ABB RAPID module: Module1.mod

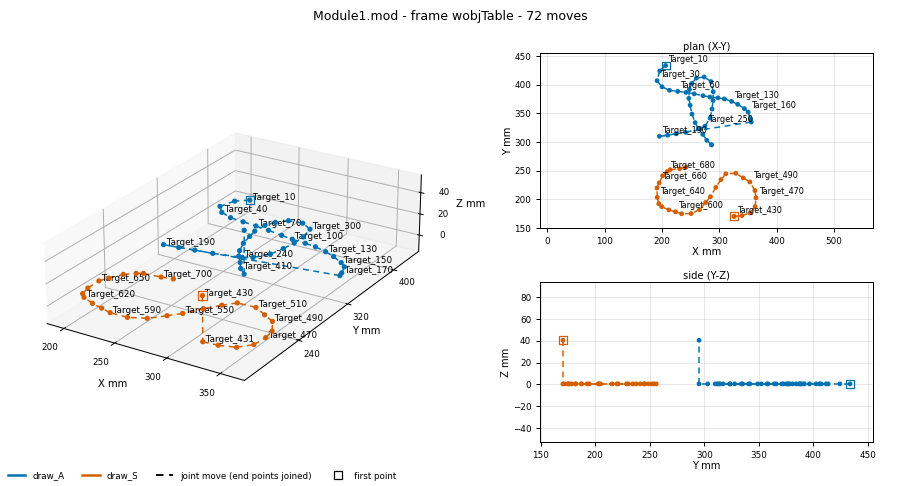
[picture p0: tool path of Module1.mod in frame wobjTable, 72 of 76 moves have a stored position in this frame; points joined in program order, loops and branches not executed]
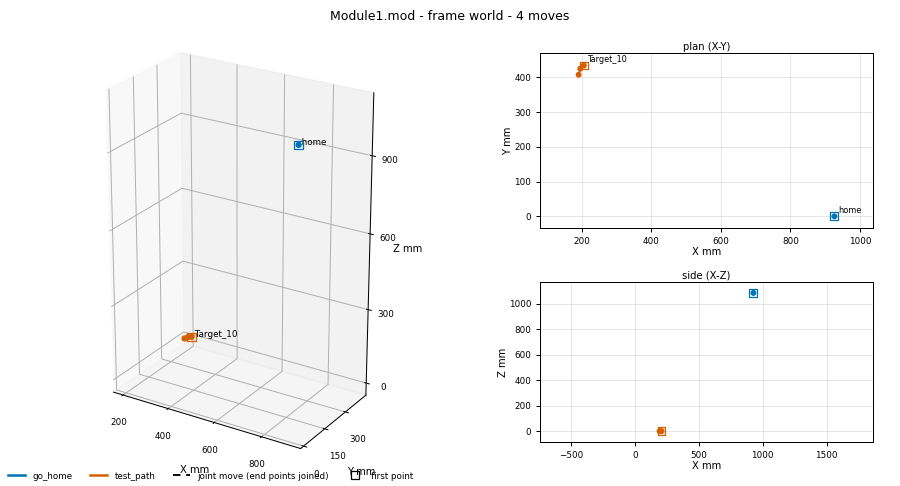
[picture p1: tool path of Module1.mod in frame world, 4 of 76 moves have a stored position in this frame; points joined in program order, loops and branches not executed]
MODULE Module1
	CONST robtarget home:=[[926.669182372,0,1084.5],[0.5,0,0.866025404,0],[0,0,0,0],[9E+09,9E+09,9E+09,9E+09,9E+09,9E+09]];
	CONST robtarget Target_10:=[[206.293,433.63,0.5],[0,0,1,0],[0,0,0,0],[9E+09,9E+09,9E+09,9E+09,9E+09,9E+09]];
	CONST robtarget Target_20:=[[196.05,424.338,0.5],[0,0,1,0],[0,0,0,0],[9E+09,9E+09,9E+09,9E+09,9E+09,9E+09]];
	CONST robtarget Target_30:=[[191.33,407.149,0.5],[0,0,1,0],[0,0,0,0],[9E+09,9E+09,9E+09,9E+09,9E+09,9E+09]];
	CONST robtarget Target_40:=[[200.077,396.45,0.5],[0,0,1,0],[0,0,0,0],[9E+09,9E+09,9E+09,9E+09,9E+09,9E+09]];
	CONST robtarget Target_50:=[[213.027,390.387,0.5],[0,0,1,0],[0,0,0,0],[9E+09,9E+09,9E+09,9E+09,9E+09,9E+09]];
	CONST robtarget Target_60:=[[227.402,388.502,0.5],[0,0,1,0],[0,0,0,0],[9E+09,9E+09,9E+09,9E+09,9E+09,9E+09]];
	CONST robtarget Target_70:=[[241.792,386.616,0.5],[0,0,1,0],[0,0,0,0],[9E+09,9E+09,9E+09,9E+09,9E+09,9E+09]];
	CONST robtarget Target_80:=[[256.194,384.262,0.5],[0,0,1,0],[0,0,0,0],[9E+09,9E+09,9E+09,9E+09,9E+09,9E+09]];
	CONST robtarget Target_90:=[[271.536,380.972,0.5],[0,0,1,0],[0,0,0,0],[9E+09,9E+09,9E+09,9E+09,9E+09,9E+09]];
	CONST robtarget Target_100:=[[283.637,378.618,0.5],[0,0,1,0],[0,0,0,0],[9E+09,9E+09,9E+09,9E+09,9E+09,9E+09]];
	CONST robtarget Target_110:=[[297.618,377.191,0.5],[0,0,1,0],[0,0,0,0],[9E+09,9E+09,9E+09,9E+09,9E+09,9E+09]];
	CONST robtarget Target_120:=[[308.809,375.301,0.5],[0,0,1,0],[0,0,0,0],[9E+09,9E+09,9E+09,9E+09,9E+09,9E+09]];
	CONST robtarget Target_130:=[[321.398,371.074,0.5],[0,0,1,0],[0,0,0,0],[9E+09,9E+09,9E+09,9E+09,9E+09,9E+09]];
	CONST robtarget Target_140:=[[332.122,365.914,0.5],[0,0,1,0],[0,0,0,0],[9E+09,9E+09,9E+09,9E+09,9E+09,9E+09]];
	CONST robtarget Target_150:=[[343.779,358.412,0.5],[0,0,1,0],[0,0,0,0],[9E+09,9E+09,9E+09,9E+09,9E+09,9E+09]];
	CONST robtarget Target_160:=[[350.301,352.321,0.5],[0,0,1,0],[0,0,0,0],[9E+09,9E+09,9E+09,9E+09,9E+09,9E+09]];
	CONST robtarget Target_170:=[[354.455,340.628,0.5],[0,0,1,0],[0,0,0,0],[9E+09,9E+09,9E+09,9E+09,9E+09,9E+09]];
	CONST robtarget Target_180:=[[355.831,335.016,0.5],[0,0,1,0],[0,0,0,0],[9E+09,9E+09,9E+09,9E+09,9E+09,9E+09]];
	CONST robtarget Target_190:=[[195.464,310.023,0.5],[0,0,1,0],[0,0,0,0],[9E+09,9E+09,9E+09,9E+09,9E+09,9E+09]];
	CONST robtarget Target_200:=[[209.832,311.96,0.5],[0,0,1,0],[0,0,0,0],[9E+09,9E+09,9E+09,9E+09,9E+09,9E+09]];
	CONST robtarget Target_210:=[[224.671,314.499,0.5],[0,0,1,0],[0,0,0,0],[9E+09,9E+09,9E+09,9E+09,9E+09,9E+09]];
	CONST robtarget Target_220:=[[241.385,317.028,0.5],[0,0,1,0],[0,0,0,0],[9E+09,9E+09,9E+09,9E+09,9E+09,9E+09]];
	CONST robtarget Target_240:=[[267.009,323.298,0.5],[0,0,1,0],[0,0,0,0],[9E+09,9E+09,9E+09,9E+09,9E+09,9E+09]];
	CONST robtarget Target_250:=[[274.99,327.846,0.5],[0,0,1,0],[0,0,0,0],[9E+09,9E+09,9E+09,9E+09,9E+09,9E+09]];
	CONST robtarget Target_260:=[[283.914,341.795,0.5],[0,0,1,0],[0,0,0,0],[9E+09,9E+09,9E+09,9E+09,9E+09,9E+09]];
	CONST robtarget Target_270:=[[287.258,357.634,0.5],[0,0,1,0],[0,0,0,0],[9E+09,9E+09,9E+09,9E+09,9E+09,9E+09]];
	CONST robtarget Target_280:=[[289.199,372.546,0.5],[0,0,1,0],[0,0,0,0],[9E+09,9E+09,9E+09,9E+09,9E+09,9E+09]];
	CONST robtarget Target_290:=[[289.278,387.93,0.5],[0,0,1,0],[0,0,0,0],[9E+09,9E+09,9E+09,9E+09,9E+09,9E+09]];
	CONST robtarget Target_300:=[[285.64,405.649,0.5],[0,0,1,0],[0,0,0,0],[9E+09,9E+09,9E+09,9E+09,9E+09,9E+09]];
	CONST robtarget Target_310:=[[273.566,413.584,0.5],[0,0,1,0],[0,0,0,0],[9E+09,9E+09,9E+09,9E+09,9E+09,9E+09]];
	CONST robtarget Target_320:=[[260.057,411.732,0.5],[0,0,1,0],[0,0,0,0],[9E+09,9E+09,9E+09,9E+09,9E+09,9E+09]];
	CONST robtarget Target_330:=[[252.101,402.428,0.5],[0,0,1,0],[0,0,0,0],[9E+09,9E+09,9E+09,9E+09,9E+09,9E+09]];
	CONST robtarget Target_340:=[[247.861,391.726,0.5],[0,0,1,0],[0,0,0,0],[9E+09,9E+09,9E+09,9E+09,9E+09,9E+09]];
	CONST robtarget Target_350:=[[246.853,376.366,0.5],[0,0,1,0],[0,0,0,0],[9E+09,9E+09,9E+09,9E+09,9E+09,9E+09]];
	CONST robtarget Target_360:=[[249.115,364.257,0.5],[0,0,1,0],[0,0,0,0],[9E+09,9E+09,9E+09,9E+09,9E+09,9E+09]];
	CONST robtarget Target_370:=[[252.292,348.884,0.5],[0,0,1,0],[0,0,0,0],[9E+09,9E+09,9E+09,9E+09,9E+09,9E+09]];
	CONST robtarget Target_380:=[[257.797,333.965,0.5],[0,0,1,0],[0,0,0,0],[9E+09,9E+09,9E+09,9E+09,9E+09,9E+09]];
	CONST robtarget Target_390:=[[263.328,323.698,0.5],[0,0,1,0],[0,0,0,0],[9E+09,9E+09,9E+09,9E+09,9E+09,9E+09]];
	CONST robtarget Target_400:=[[271.19,313.417,0.5],[0,0,1,0],[0,0,0,0],[9E+09,9E+09,9E+09,9E+09,9E+09,9E+09]];
	CONST robtarget Target_410:=[[278.124,303.135,0.5],[0,0,1,0],[0,0,0,0],[9E+09,9E+09,9E+09,9E+09,9E+09,9E+09]];
	CONST robtarget Target_420:=[[286.472,295.172,0.5],[0,0,1,0],[0,0,0,0],[9E+09,9E+09,9E+09,9E+09,9E+09,9E+09]];
	CONST robtarget Target_421:=[[286.472,295.172,40.5],[0,0,1,0],[0,0,0,0],[9E+09,9E+09,9E+09,9E+09,9E+09,9E+09]];
	CONST robtarget Target_430:=[[325.977,170.345,40.5],[0,0,1,0],[0,0,0,0],[9E+09,9E+09,9E+09,9E+09,9E+09,9E+09]];
	CONST robtarget Target_431:=[[325.977,170.345,0.5],[0,0,1,0],[0,0,0,0],[9E+09,9E+09,9E+09,9E+09,9E+09,9E+09]];
	CONST robtarget Target_440:=[[339.546,171.622,0.5],[0,0,1,0],[0,0,0,0],[9E+09,9E+09,9E+09,9E+09,9E+09,9E+09]];
	CONST robtarget Target_450:=[[353.612,176.166,0.5],[0,0,1,0],[0,0,0,0],[9E+09,9E+09,9E+09,9E+09,9E+09,9E+09]];
	CONST robtarget Target_460:=[[362.57,187.303,0.5],[0,0,1,0],[0,0,0,0],[9E+09,9E+09,9E+09,9E+09,9E+09,9E+09]];
	CONST robtarget Target_470:=[[364.055,202.715,0.5],[0,0,1,0],[0,0,0,0],[9E+09,9E+09,9E+09,9E+09,9E+09,9E+09]];
	CONST robtarget Target_480:=[[362.245,215.349,0.5],[0,0,1,0],[0,0,0,0],[9E+09,9E+09,9E+09,9E+09,9E+09,9E+09]];
	CONST robtarget Target_490:=[[353.422,230.367,0.5],[0,0,1,0],[0,0,0,0],[9E+09,9E+09,9E+09,9E+09,9E+09,9E+09]];
	CONST robtarget Target_500:=[[341.755,237.455,0.5],[0,0,1,0],[0,0,0,0],[9E+09,9E+09,9E+09,9E+09,9E+09,9E+09]];
	CONST robtarget Target_510:=[[328.7,245.481,0.5],[0,0,1,0],[0,0,0,0],[9E+09,9E+09,9E+09,9E+09,9E+09,9E+09]];
	CONST robtarget Target_520:=[[311.408,244.662,0.5],[0,0,1,0],[0,0,0,0],[9E+09,9E+09,9E+09,9E+09,9E+09,9E+09]];
	CONST robtarget Target_530:=[[302.952,234.456,0.5],[0,0,1,0],[0,0,0,0],[9E+09,9E+09,9E+09,9E+09,9E+09,9E+09]];
	CONST robtarget Target_540:=[[294.019,220.996,0.5],[0,0,1,0],[0,0,0,0],[9E+09,9E+09,9E+09,9E+09,9E+09,9E+09]];
	CONST robtarget Target_550:=[[284.61,204.751,0.5],[0,0,1,0],[0,0,0,0],[9E+09,9E+09,9E+09,9E+09,9E+09,9E+09]];
	CONST robtarget Target_560:=[[276.17,194.566,0.5],[0,0,1,0],[0,0,0,0],[9E+09,9E+09,9E+09,9E+09,9E+09,9E+09]];
	CONST robtarget Target_570:=[[265.396,182.078,0.5],[0,0,1,0],[0,0,0,0],[9E+09,9E+09,9E+09,9E+09,9E+09,9E+09]];
	CONST robtarget Target_580:=[[250.937,175.221,0.5],[0,0,1,0],[0,0,0,0],[9E+09,9E+09,9E+09,9E+09,9E+09,9E+09]];
	CONST robtarget Target_590:=[[234.203,174.906,0.5],[0,0,1,0],[0,0,0,0],[9E+09,9E+09,9E+09,9E+09,9E+09,9E+09]];
	CONST robtarget Target_600:=[[223.54,178.258,0.5],[0,0,1,0],[0,0,0,0],[9E+09,9E+09,9E+09,9E+09,9E+09,9E+09]];
	CONST robtarget Target_610:=[[211.957,181.616,0.5],[0,0,1,0],[0,0,0,0],[9E+09,9E+09,9E+09,9E+09,9E+09,9E+09]];
	CONST robtarget Target_620:=[[199.469,187.304,0.5],[0,0,1,0],[0,0,0,0],[9E+09,9E+09,9E+09,9E+09,9E+09,9E+09]];
	CONST robtarget Target_630:=[[194.398,192.459,0.5],[0,0,1,0],[0,0,0,0],[9E+09,9E+09,9E+09,9E+09,9E+09,9E+09]];
	CONST robtarget Target_640:=[[191.676,203.634,0.5],[0,0,1,0],[0,0,0,0],[9E+09,9E+09,9E+09,9E+09,9E+09,9E+09]];
	CONST robtarget Target_650:=[[191.297,219.9,0.5],[0,0,1,0],[0,0,0,0],[9E+09,9E+09,9E+09,9E+09,9E+09,9E+09]];
	CONST robtarget Target_660:=[[195.047,228.701,0.5],[0,0,1,0],[0,0,0,0],[9E+09,9E+09,9E+09,9E+09,9E+09,9E+09]];
	CONST robtarget Target_670:=[[201.135,241.207,0.5],[0,0,1,0],[0,0,0,0],[9E+09,9E+09,9E+09,9E+09,9E+09,9E+09]];
	CONST robtarget Target_680:=[[209.054,248.593,0.5],[0,0,1,0],[0,0,0,0],[9E+09,9E+09,9E+09,9E+09,9E+09,9E+09]];
	CONST robtarget Target_690:=[[214.172,251.815,0.5],[0,0,1,0],[0,0,0,0],[9E+09,9E+09,9E+09,9E+09,9E+09,9E+09]];
	CONST robtarget Target_700:=[[230.89,253.569,0.5],[0,0,1,0],[0,0,0,0],[9E+09,9E+09,9E+09,9E+09,9E+09,9E+09]];
	CONST robtarget Target_710:=[[241.587,255.829,0.5],[0,0,1,0],[0,0,0,0],[9E+09,9E+09,9E+09,9E+09,9E+09,9E+09]];
    !***********************************************************
    !
    ! Module:  Module1
    !
    ! Description:
    !   <Insert description here>
    !
    ! Author: user
    !
    ! Version: 1.0
    !
    !***********************************************************


    !***********************************************************
    !
    ! Procedure main
    !
    !   This is the entry point of your program
    !
    !***********************************************************
    PROC main()
		go_home;
		test_path;
		draw_A;
		draw_S;
		go_home;
        !Add your code here
    ENDPROC
	PROC go_home()
	    MoveJ home,v100,fine,pen\WObj:=wobj0;
	ENDPROC
	PROC test_path()
	    MoveJ Target_10,v100,fine,pen\WObj:=wobj0;
	    MoveJ Target_20,v100,fine,pen\WObj:=wobj0;
	    MoveJ Target_30,v100,fine,pen\WObj:=wobj0;
	ENDPROC
	PROC draw_A()
	    MoveJ Target_10,v100,fine,pen\WObj:=wobjTable;
	    MoveJ Target_20,v100,fine,pen\WObj:=wobjTable;
	    MoveJ Target_30,v100,fine,pen\WObj:=wobjTable;
	    MoveJ Target_40,v100,fine,pen\WObj:=wobjTable;
	    MoveJ Target_50,v100,fine,pen\WObj:=wobjTable;
	    MoveJ Target_60,v100,fine,pen\WObj:=wobjTable;
	    MoveJ Target_70,v100,fine,pen\WObj:=wobjTable;
	    MoveJ Target_80,v100,fine,pen\WObj:=wobjTable;
	    MoveJ Target_90,v100,fine,pen\WObj:=wobjTable;
	    MoveJ Target_100,v100,fine,pen\WObj:=wobjTable;
	    MoveJ Target_110,v100,fine,pen\WObj:=wobjTable;
	    MoveJ Target_120,v100,fine,pen\WObj:=wobjTable;
	    MoveJ Target_130,v100,fine,pen\WObj:=wobjTable;
	    MoveJ Target_140,v100,fine,pen\WObj:=wobjTable;
	    MoveJ Target_150,v100,fine,pen\WObj:=wobjTable;
	    MoveJ Target_160,v100,fine,pen\WObj:=wobjTable;
	    MoveJ Target_170,v100,fine,pen\WObj:=wobjTable;
	    MoveJ Target_180,v100,fine,pen\WObj:=wobjTable;
	    MoveJ Target_190,v100,fine,pen\WObj:=wobjTable;
	    MoveJ Target_200,v100,fine,pen\WObj:=wobjTable;
	    MoveJ Target_210,v100,fine,pen\WObj:=wobjTable;
	    MoveJ Target_220,v100,fine,pen\WObj:=wobjTable;
	    MoveJ Target_240,v100,fine,pen\WObj:=wobjTable;
	    MoveJ Target_250,v100,fine,pen\WObj:=wobjTable;
	    MoveJ Target_260,v100,fine,pen\WObj:=wobjTable;
	    MoveJ Target_270,v100,fine,pen\WObj:=wobjTable;
	    MoveJ Target_280,v100,fine,pen\WObj:=wobjTable;
	    MoveJ Target_290,v100,fine,pen\WObj:=wobjTable;
	    MoveJ Target_300,v100,fine,pen\WObj:=wobjTable;
	    MoveJ Target_310,v100,fine,pen\WObj:=wobjTable;
	    MoveJ Target_320,v100,fine,pen\WObj:=wobjTable;
	    MoveJ Target_330,v100,fine,pen\WObj:=wobjTable;
	    MoveJ Target_340,v100,fine,pen\WObj:=wobjTable;
	    MoveJ Target_350,v100,fine,pen\WObj:=wobjTable;
	    MoveJ Target_360,v100,fine,pen\WObj:=wobjTable;
	    MoveJ Target_370,v100,fine,pen\WObj:=wobjTable;
	    MoveJ Target_380,v100,fine,pen\WObj:=wobjTable;
	    MoveJ Target_390,v100,fine,pen\WObj:=wobjTable;
	    MoveJ Target_400,v100,fine,pen\WObj:=wobjTable;
	    MoveJ Target_410,v100,fine,pen\WObj:=wobjTable;
	    MoveJ Target_420,v100,fine,pen\WObj:=wobjTable;
	    MoveJ Target_421,v100,fine,pen\WObj:=wobjTable;
	ENDPROC
	PROC draw_S()
	    MoveJ Target_430,v100,fine,pen\WObj:=wobjTable;
	    MoveJ Target_431,v100,fine,pen\WObj:=wobjTable;
	    MoveJ Target_440,v100,fine,pen\WObj:=wobjTable;
	    MoveJ Target_450,v100,fine,pen\WObj:=wobjTable;
	    MoveJ Target_460,v100,fine,pen\WObj:=wobjTable;
	    MoveJ Target_470,v100,fine,pen\WObj:=wobjTable;
	    MoveJ Target_480,v100,fine,pen\WObj:=wobjTable;
	    MoveJ Target_490,v100,fine,pen\WObj:=wobjTable;
	    MoveJ Target_500,v100,fine,pen\WObj:=wobjTable;
	    MoveJ Target_510,v100,fine,pen\WObj:=wobjTable;
	    MoveJ Target_520,v100,fine,pen\WObj:=wobjTable;
	    MoveJ Target_530,v100,fine,pen\WObj:=wobjTable;
	    MoveJ Target_540,v100,fine,pen\WObj:=wobjTable;
	    MoveJ Target_550,v100,fine,pen\WObj:=wobjTable;
	    MoveJ Target_560,v100,fine,pen\WObj:=wobjTable;
	    MoveJ Target_570,v100,fine,pen\WObj:=wobjTable;
	    MoveJ Target_580,v100,fine,pen\WObj:=wobjTable;
	    MoveJ Target_590,v100,fine,pen\WObj:=wobjTable;
	    MoveJ Target_600,v100,fine,pen\WObj:=wobjTable;
	    MoveJ Target_610,v100,fine,pen\WObj:=wobjTable;
	    MoveJ Target_620,v100,fine,pen\WObj:=wobjTable;
	    MoveJ Target_630,v100,fine,pen\WObj:=wobjTable;
	    MoveJ Target_640,v100,fine,pen\WObj:=wobjTable;
	    MoveJ Target_650,v100,fine,pen\WObj:=wobjTable;
	    MoveJ Target_660,v100,fine,pen\WObj:=wobjTable;
	    MoveJ Target_670,v100,fine,pen\WObj:=wobjTable;
	    MoveJ Target_680,v100,fine,pen\WObj:=wobjTable;
	    MoveJ Target_690,v100,fine,pen\WObj:=wobjTable;
	    MoveJ Target_700,v100,fine,pen\WObj:=wobjTable;
	    MoveJ Target_710,v100,fine,pen\WObj:=wobjTable;
	ENDPROC
ENDMODULE
